{attribute addProperty BoxType "EP9214-0023-0019"}
{attribute addProperty Id "Output_UsAT %Q*BOOL811Output_UpAT %Q*BOOL812Reset_UsAT %Q*BOOL815Reset_UpAT %Q*BOOL816"}
{attribute addProperty CRC "1465931327"}
{attribute addProperty SizeInBites "32"}
{attribute addProperty SizeInBytes "4"}
TYPE DPO_Outputs_Channel_5760563F :
STRUCT
	{attribute addProperty Name "Output_Us"}
	Output_Us AT %Q* : BOOL;
	{attribute addProperty Name "Output_Up"}
	Output_Up AT %Q* : BOOL;
	{attribute addProperty Name "Reset_Us"}
	Reset_Us AT %Q* : BOOL;
	{attribute addProperty Name "Reset_Up"}
	Reset_Up AT %Q* : BOOL;
END_STRUCT
END_TYPE

(* stored: Version 1.2.0.0, ProductVersion 3.1.4024.9
   DUT DPO_Outputs_Channel_5760563F: Id {c08dba44-bae1-4922-80b5-c52c7b407254} *)
